(* PLC project SansNom, Inconnu SansNom 1 *)
(* stored: creationDateTime 2025-01-20T19:01:41, modificationDateTime 2025-01-21T09:51:17 *)

PROGRAM program0
  VAR
    Test1 : INT;
    Test2 : INT;
    Test3 : BOOL;
    Test0 : Test;
  END_VAR

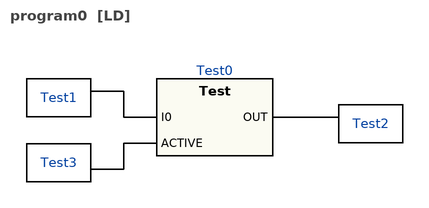
(* LD diagram, written out as Structured Text *)
Test0(I0 := Test1, ACTIVE := Test3);
Test2 := Test0.OUT;
END_PROGRAM

CONFIGURATION Config0
  RESOURCE Res0 ON PLC
    TASK task0(INTERVAL := T#20ms, PRIORITY := 0);
    PROGRAM instance0 WITH task0 : program0;
  END_RESOURCE
END_CONFIGURATION
